FUNCTION_BLOCK "abb_aquaMaster_3"
{ S7_Optimized_Access := 'TRUE' }
VERSION : 0.1
   VAR_INPUT
      mb_addr : USInt;
   END_VAR

   VAR_IN_OUT
      mb_query : "mb_query";
   END_VAR

   VAR
      s : "mb_station_udt";
      flow : Real;
      pressure : Real;
      totaliser : Struct
         fwd : DInt;
         rev : DInt;
         net : DInt;
      END_STRUCT;
   END_VAR


BEGIN
	// - ABB - AquaMaster 3 - Electromagnetic flowmeter
	// - COI/FET2XX/MOD/TBLâ€“EN
	// - https://library.e.abb.com/public/
	//   91eead459bb0d349c12577fc0033d2b5/COI_FET2XX_MOD_TBL-EN.pdf

	"mb_station_header"(station := #s, mb_query := #mb_query);
	#mb_query.mb_addr := #mb_addr; // Device address.

	// Two queries, reading input registers.
	#mb_query.mode := #mb_query.c.read.input_reg;
	#mb_query(data_addr := 5017, data_ptr := #flow);
	#mb_query(data_addr := 5025, data_ptr := #pressure);

	// One query, reading one section of holding registers.
	#mb_query.mode := #mb_query.c.read.holding_reg;
	#mb_query(data_addr := 12003, data_ptr := #totaliser );

	// - Each query reading one section of holding registers.
	// - Data length is automatically calculated for holding
	//   and input regisers.
	// - mb_query_bits should be used for discrete in- and outpus.

	"mb_station_footer"(station := #s, mb_query := #mb_query);

END_FUNCTION_BLOCK

FUNCTION_BLOCK "start_example_modbus_rtu"
{ S7_Optimized_Access := 'TRUE' }
VERSION : 0.1
   VAR
      mb_query : "mb_query";
      mb_master_ctrl : "mb_master_1200_ctrl";
      abb_aquaMaster_device1 : "abb_aquaMaster_3";
      abb_aquaMaster_device2 : "abb_aquaMaster_3";
      abb_aquaMaster_device3 : "abb_aquaMaster_3";
      resault_data_1 : Word;
   END_VAR


BEGIN
	// This a rtu example for S7-1200, for S7-1500 use
	// mb_master_1500_ctrl.

	// hardware_id: Can be found inside the hardware configuration.
	// baud:        bps. (parity is even by default)
	// timeout:     Automatically calculated if not specified.
	// mb_query:    A FB.
	#mb_master_ctrl(hardware_id := "Local~CB_1241_(RS485)",
	                baud := 19200,
	                mb_query := #mb_query);

	// In this rtu example there are 3 devices connected to the
	// modbus-rtu bus. Each instance of the blocks bellow represent one
	// device on the bus. A "station block" has to be created for each
	// spesific modbus device.

	// Three abb aqua-master's.
	#abb_aquaMaster_device1(mb_addr := 1, mb_query := #mb_query);
	#abb_aquaMaster_device2(mb_addr := 2, mb_query := #mb_query);
	#abb_aquaMaster_device3(mb_addr := 3, mb_query := #mb_query);

	// Keep in mind that a station block can be used both for both modbus
	// rtu and tcp. This is specially useful if a tcp-rtu-gateway is used.
	// The same program could be used, just swap mb_master_ctrl, with
	// mb_client_ctrl.


	// Read holding register 456 (zero counted) from device with modbus
	// address 123. This is an example showing that a query does not
	// necessarily need to be part of a station block (SB) as obove, however
	// making reusable SB's is good practice.
	#mb_query(mb_addr := 123,
	          mode := #mb_query.c.read.holding_reg,
	          data_addr := 456,
	          data_ptr := #resault_data_1);

END_FUNCTION_BLOCK

DATA_BLOCK "start_example_modbus_rtu_DB"
{ S7_Optimized_Access := 'TRUE' }
VERSION : 0.1
NON_RETAIN
"start_example_modbus_rtu"

BEGIN

END_DATA_BLOCK

ORGANIZATION_BLOCK "rtu_ob"
TITLE = "Main Program Sweep (Cycle)"
{ S7_Optimized_Access := 'TRUE' }
VERSION : 0.1

BEGIN
	// Program cycle OB

	// Open the block to see the example.
	"start_example_modbus_rtu_DB"();

END_ORGANIZATION_BLOCK

